Staubli VAL3: Step1.pjx

--- Step1.pjx ---
Parameters version=s7.9.1 stackSize=5000 millimeterUnit=true
Program file=ConstuireMur.pgx
Program file=ConstuireSol.pgx
Program file=OpenPince_test.pgx
Program file=saisirpiecev1.pgx
Program file=start.pgx
Program file=stop.pgx
Program file=test_decoupe.pgx
Program file=testDonneCall.pgx
Program file=Tour.pgx
Data file=Step1.dtx

--- Step1.dtx ---
mdesc mNomSpeed
pointRx Starting_point = {x=-380, y=80, z=150, rx=180, rz=-90, fatherId=world[0]}
pointRx Real_start = {fatherId=world[0]}
pointRx B = {rx=180, fatherId=world[0]}
pointRx C = {rx=180, fatherId=world[0]}
pointRx D = {rx=180, fatherId=world[0]}
pointRx E = {rx=180, fatherId=world[0]}
num Dim_width
num Dim_height
screen sEcran
num nYN
num nx
num ny
num nz
num nRx
num nRy
num nRz
tool tTool = {fatherId=flange[0], ioLink=valve1}
pointRx pCentrepiece1[4]
  [0] = {x=-170, y=-290, rx=180, rz=-90, fatherId=world[0]}
  [1] = {x=-56, y=-290, rx=180, rz=-90, fatherId=world[0]}
  [2] = {x=58, y=-290, rx=180, rz=-90, fatherId=world[0]}
  [3] = {x=170, y=-290, rx=180, rz=-90, fatherId=world[0]}
num nNbPieceMax = 6
num nNbPieceArrive
pointRx Real_Stop = {fatherId=world[0]}
pointRx pCentre_Arrive[7]
  [0] = {y=335, rx=180, fatherId=world[0]}
  [1] = {y=240, rx=180, fatherId=world[0]}
  [2] = {x=50, y=290, rx=180, rz=90, fatherId=world[0]}
  [3] = {x=-50, y=290, rx=180, rz=90, fatherId=world[0]}
  [4] = {x=-20, y=290, rx=180, rz=90, fatherId=world[0]}
  [5] = {x=20, y=290, rx=180, rz=90, fatherId=world[0]}
  [6] = {y=290, z=150, rx=180, fatherId=world[0]}
pointRx pTestTemp = {y=-290, z=-180, rx=180, fatherId=world[0]}
pointRx B_haut = {fatherId=world[0]}
num i
num nNbEtage
num DepotStock[4]
  [0] = 5
  [1] = 5
  [2] = 5
  [3] = 5
num indiceStock
num nValeurAngle

--- start.pgx ---
program start()
begin
   userPage(sEcran)
  cls(sEcran)
   putln(sEcran, "Quel programme voulez vous lancer : ")
  putln(sEcran, "   1. Découpe")
  putln(sEcran, "   2. Tour de 4 pièces")
  putln(sEcran, "   3. Constuire tour")
  get(sEcran, nYN)
  if nYN == 1
    call test_decoupe()
  elseIf nYN==2
    call saisirpiecev1()
  elseIf nYN==3
    call Tour()
  endIf
end

--- ConstuireMur.pgx ---
program ConstuireMur()
begin

  userPage(sEcran)
  cls(sEcran)

  //on va a la position de depart
   movej(Starting_point, tTool, mNomSpeed)
  waitEndMove()
  //on ouvre la pince
  open(tTool)

  for i = 0 to 3
    //on prend le depot ou il y a des pièces en stock
    while(DepotStock[indiceStock]<1)
      indiceStock=indiceStock+1
    endWhile

    //on vas au dessus de la zone à saisir
    //pCentrePiece est un tableau qui contient les position au dessus des stocks
    Real_start=pCentrepiece1[indiceStock]
    //note:plus z est grand plus le bras sera haut
    //la on est au dessus
    movej(Real_start, tTool, mNomSpeed)
    waitEndMove()

    //on vas a la piece on met le 123 pour descendre sinon on est trop haut
    B = {{Real_start.trsf.x , Real_start.trsf.y, Real_start.trsf.z-180+(DepotStock[indiceStock])*7, Real_start.trsf.rx, Real_start.trsf.ry, Real_start.trsf.rz}, {sfree, efree, wfree}}
    movel(B, tTool, mNomSpeed)
    waitEndMove()
    //on ferme la pince
    close(tTool)
    //on revient au dessus
    movel(Real_start, tTool, mNomSpeed)
    waitEndMove()

    //Real_Stop=pCentre_Arrive

    //on amene la piece au dessus de la position où construire
    //pCentre_Arrive contient un tableau avec les 6 positions possibles de depots
    movej(pCentre_Arrive[6], tTool, mNomSpeed)
    waitEndMove()
   //on baisse la pince
    Real_Stop = {{pCentre_Arrive[i].trsf.x , pCentre_Arrive[i].trsf.y, pCentre_Arrive[i].trsf.z-165+nNbEtage*10, pCentre_Arrive[i].trsf.rx, pCentre_Arrive[i].trsf.ry, pCentre_Arrive[i].trsf.rz}, {sfree, efree, wfree}}

     //on modifi l'angle si necessaire
     if i >1
      Real_Stop.trsf.rz=Real_start.trsf.rz+nValeurAngle
    endIf

    movel(Real_Stop, tTool, mNomSpeed)
    waitEndMove()
    //on ouvre la pince
    open(tTool)
    //on relève la pince
    movel(pCentre_Arrive[6], tTool, mNomSpeed)
    waitEndMove()
    DepotStock[indiceStock]=DepotStock[indiceStock]-1
    if i==1
      nNbEtage=nNbEtage+1
    endIf
  endFor

  //on retourne à la position de départ
  movej(Starting_point, tTool, mNomSpeed)
  waitEndMove()
 //on ferme la pince
close(tTool)

  put(sEcran, "Operation réalisé")
end

--- ConstuireSol.pgx ---
program ConstuireSol()
begin

  userPage(sEcran)
  cls(sEcran)

  //on va a la position de depart
   movej(Starting_point, tTool, mNomSpeed)
  waitEndMove()
  //on ouvre la pince
  open(tTool)

  for i = 0 to 5
    //on prend le depot ou il y a des pièces en stock
    while(DepotStock[indiceStock]<1)
      indiceStock=indiceStock+1
    endWhile

    //on vas au dessus de la zone à saisir
    //pCentrePiece est un tableau qui contient les position au dessus des stocks
    Real_start=pCentrepiece1[indiceStock]

    //note:plus z est grand plus le bras sera haut
    //la on est au dessus
    movej(Real_start, tTool, mNomSpeed)
    waitEndMove()

    //on vas a la piece on met le 123 pour descendre sinon on est trop haut
    B = {{Real_start.trsf.x , Real_start.trsf.y, Real_start.trsf.z-180+(DepotStock[indiceStock])*7, Real_start.trsf.rx, Real_start.trsf.ry, Real_start.trsf.rz}, {sfree, efree, wfree}}
    movel(B, tTool, mNomSpeed)
    waitEndMove()
    //on ferme la pince
    close(tTool)
    //on revient au dessus
    movel(Real_start, tTool, mNomSpeed)
    waitEndMove()

    //Real_Stop=pCentre_Arrive

    //on amene la piece au dessus de la position où construire
    //pCentre_Arrive contient un tableau avec les 6 positions possibles de depots
    movej(pCentre_Arrive[6], tTool, mNomSpeed)
    waitEndMove()


   //on baisse la pince
    Real_Stop = {{pCentre_Arrive[i].trsf.x , pCentre_Arrive[i].trsf.y, pCentre_Arrive[i].trsf.z-165+nNbEtage*10, pCentre_Arrive[i].trsf.rx, pCentre_Arrive[i].trsf.ry, pCentre_Arrive[i].trsf.rz}, {sfree, efree, wfree}}
     //on modifi l'angle si necessaire
     if i >1
      Real_Stop.trsf.rz=Real_start.trsf.rz+nValeurAngle
    endIf

    movel(Real_Stop, tTool, mNomSpeed)
    waitEndMove()
    //on ouvre la pince
    open(tTool)
    //on relève la pince
    movel(pCentre_Arrive[6], tTool, mNomSpeed)
    waitEndMove()
    DepotStock[indiceStock]=DepotStock[indiceStock]-1
    if i==1
      nNbEtage=nNbEtage+1
    endIf
  endFor

  //on retourne à la position de départ
  movej(Starting_point, tTool, mNomSpeed)
  waitEndMove()
 //on ferme la pince
close(tTool)

  put(sEcran, "Operation réalisé")
end

--- OpenPince_test.pgx ---
program OpenPince_test()
begin

  userPage(sEcran)
  cls(sEcran)

  close(tTool)
  open(tTool)
    put(sEcran, "Operation réalisé")
end

--- saisirpiecev1.pgx ---
program saisirpiecev1()
begin

  userPage(sEcran)
  cls(sEcran)

  //on va a la position de depart
   movej(Starting_point, tTool, mNomSpeed)
  waitEndMove()
  //on ouvre la pince
    open(tTool)
  for i = 0 to 3

    //on vas au dessus de la zone à saisir
    Real_start=pCentrepiece1[1]
    //note:plus z est grand plus le bras sera haut
    //la on est au dessus
    movej(Real_start, tTool, mNomSpeed)
    waitEndMove()

    //on vas a la piece on met le 123 pour descendre sinon on est trop haut
    B = {{Real_start.trsf.x , Real_start.trsf.y, Real_start.trsf.z-180+(DepotStock[1])*7, Real_start.trsf.rx, Real_start.trsf.ry, Real_start.trsf.rz}, {sfree, efree, wfree}}
    movel(B, tTool, mNomSpeed)
    waitEndMove()
    //on ferme la pince
    close(tTool)
    //on revient au dessus
    movel(Real_start, tTool, mNomSpeed)
    waitEndMove()

    //Real_Stop=pCentre_Arrive

    //on amene la piece au dessus de la position où construire
    movej(pCentre_Arrive[6], tTool, mNomSpeed)
    waitEndMove()
   //on baisse la pince
    Real_Stop = {{pCentre_Arrive[0].trsf.x , pCentre_Arrive[0].trsf.y, pCentre_Arrive[0].trsf.z-165+nNbEtage*7, pCentre_Arrive[0].trsf.rx, pCentre_Arrive[0].trsf.ry, pCentre_Arrive[0].trsf.rz}, {sfree, efree, wfree}}
    movel(Real_Stop, tTool, mNomSpeed)
    waitEndMove()
    //on ouvre la pince
    open(tTool)
    //on relève la pince
    movel(pCentre_Arrive[6], tTool, mNomSpeed)
    waitEndMove()
    DepotStock[1]=DepotStock[1]-1
    nNbEtage=nNbEtage+1
  endFor

  //on retourne à la position de départ
  movej(Starting_point, tTool, mNomSpeed)
  waitEndMove()
 //on ferme la pince
close(tTool)

  put(sEcran, "Operation réalisé")
end

--- test_decoupe.pgx ---
program test_decoupe()
begin

  userPage(sEcran)
  cls(sEcran)
  //on vas à la position initiale

  movej(Starting_point, tTool, mNomSpeed)
  waitEndMove()

  //	demande si point de départ custo
  putln(sEcran, "Voulez vous changer le point de départ de la découpe : ")
  putln(sEcran, "   1. Oui")
  putln(sEcran, "   2. Non")
  get(sEcran, nYN)
  //	si oui recuperation
  if nYN == 1
    putln(sEcran, "x = ")
    get(sEcran, nx)

    putln(sEcran, "y = ")
    get(sEcran, ny)

    putln(sEcran, "z = ")
    get(sEcran, nz)

    putln(sEcran, "Rx = ")
    get(sEcran, nRx)

    putln(sEcran, "Ry = ")
    get(sEcran, nRy)

    putln(sEcran, "Rz = ")
    get(sEcran, nRz)

    Real_start = {{nx,ny,nz,nRx,nRy,nRz}, {sfree, efree, wfree}}
  else
    //	sinon point de depart par defaut
    Real_start=Starting_point
  endIf

  //récupération largeur et hauteur de la découpe:
  //	demande si dimension custo
  putln(sEcran, "Voulez vous changer les dimensions de la découpe : ")
  putln(sEcran, "   1. Oui")
  putln(sEcran, "   2. Non")
  get(sEcran, nYN)
  if nYN == 1
  //	si oui recuperation
  putln(sEcran, "")
  putln(sEcran, "Veuillez entrer les dimensions de votre découpe :")

  put(sEcran, "Hauteur = ")
  get(sEcran, Dim_height)
  put(sEcran, Dim_height)
  putln(sEcran, "")

  put(sEcran, "Largeur = ")
  get(sEcran, Dim_width)
  put(sEcran, Dim_width)
  putln(sEcran, "")
  else
    //	sinon demension par defaut
    Dim_height = 5
    Dim_width = 10
  endIf

  //découpe (par defaut on comence en haut à gauche)
  B = {{Real_start.trsf.x - Dim_height/2, Real_start.trsf.y + Dim_height/2, Real_start.trsf.z, Real_start.trsf.rx, Real_start.trsf.ry, Real_start.trsf.rz}, {sfree, efree, wfree}}
  C = {{Real_start.trsf.x - Dim_height, Real_start.trsf.y, Real_start.trsf.z, Real_start.trsf.rx, Real_start.trsf.ry, Real_start.trsf.rz}, {sfree, efree, wfree}}
  D = {{Real_start.trsf.x - Dim_height, Real_start.trsf.y + Dim_width, Real_start.trsf.z, Real_start.trsf.rx, Real_start.trsf.ry, Real_start.trsf.rz}, {sfree, efree, wfree}}
  E = {{Real_start.trsf.x, Real_start.trsf.y + Dim_width, Real_start.trsf.z, Real_start.trsf.rx, Real_start.trsf.ry, Real_start.trsf.rz}, {sfree, efree, wfree}}


  movel(Real_start, tTool, mNomSpeed)
  waitEndMove()

  movec(B,C,tTool, mNomSpeed)
  waitEndMove()

  movel(D, tTool, mNomSpeed)
  waitEndMove()

  movel(E, tTool, mNomSpeed)
  waitEndMove()

  movel(Real_start, tTool, mNomSpeed)
  waitEndMove()

  //on vas à la position initiale
  movej(Starting_point, tTool, mNomSpeed)
  waitEndMove()

  put(sEcran, "Operation réalisé")
end

--- testDonneCall.pgx ---
program testDonneCall()
begin
  putln(sEcran,nNbPieceArrive)
end

--- Tour.pgx ---
program Tour()
begin

  userPage(sEcran)
  cls(sEcran)
  while (DepotStock[0]+DepotStock[1]+DepotStock[2]+DepotStock[3]>3)
    putln(sEcran, "Voulez vous creer : ")
    putln(sEcran, "   1. Creer un Mur 4 pieces")
    putln(sEcran, "   2. Creer un Sol 6 pièces")
    putln(sEcran, "   3. Modifier l'angle")
    put(sEcran, "Il reste ")
    put(sEcran, DepotStock[0]+DepotStock[1]+DepotStock[2]+DepotStock[3])
    putln(sEcran, " pièces ")
    get(sEcran, nYN)
    //pour simplifier on vas vider les dépots 1 par 1
    if nYN == 1
      call ConstuireMur()
    elseIf nYN==2
      call ConstuireSol()
    else
      putln(sEcran, "   Entrer la valeur de l'angle (0 par défaut)")
      get(sEcran, nValeurAngle)
    endIf
    nNbEtage=nNbEtage+1
  endWhile
end
